// TIA Portal V20 export
DATA_BLOCK "BK20"   // DB311
// stored: MemoryReserve 100
   VAR
      "X10-1.STACK TABLE Z-AXIS LIMIT SENSOR(-)" : Bool := TRUE;
      "X11-1.STACK TABLE Z-AXIS LIMIT SENSOR(+)" : Bool := TRUE;
      "X12-1.STACK TABLE GAP PAD DOWN" : Bool := TRUE;
      "X13-1.STACK TABLE GAP PAD UP" : Bool := FALSE;
      "X14-1.STACK TABLE OUT FRONT Z-AXIS LIMIT SENSOR(-)" : Bool := TRUE;
      "X15-1.STACK TABLE OUT FRONT Z-AXIS LIMIT SENSOR(+)" : Bool := TRUE;
      "X16-1.STACK TABLE VACUUM PRESSURE SWITCH" : Bool := FALSE;
      "X17-1.SPARE" : Bool := FALSE;
      "X10-2.STACK TABLE Z-AXIS HOME SENSOR" : Bool := TRUE;
      "X11-2.SPARE" : Bool := FALSE;
      "X12-2.SPARE" : Bool := FALSE;
      "X13-2.SPARE" : Bool := FALSE;
      "X14-2.STACK TABLE OUT FRONT Z-AXIS HOME SENSOR" : Bool := TRUE;
      "X15-2.SPARE" : Bool := FALSE;
      "X16-2.STACK TABLE ELECTRODE DETECT SENSOR" : Bool := FALSE;
      "X17-2.SPARE" : Bool := FALSE;
   END_VAR
BEGIN
END_DATA_BLOCK
